// TIA Portal V16 export
// export: Created 2024-09-05T17:40:14.5392441Z, ExportSetting WithDefaults, DisplayName Totally Integrated Automation Portal, DisplayVersion V16 Update 6, DisplayName TIA Portal Version Control Interface, DisplayVersion V16 Update 2, DisplayName TIA Portal Openness, DisplayVersion V16 Update 6, DisplayName STEP 7 Professional, DisplayVersion V16 Update 6, DisplayName STEP 7 Safety, DisplayVersion V16, DisplayName WinCC Advanced, DisplayVersion V16 Update 6
TYPE "UDT_Friedrich"
// stored: IsFailsafeCompliant false
   STRUCT
      Start : Bool;
      PrgNumber : Int;
      Ready : Bool;
      Running : Bool;
      OK : Bool;
      NOK : Bool;
      H1OK : Bool;
      H2OK : Bool;
      TimeOK : Bool;
      StartError : Bool;
      LastH1 : Real;
      LastH2 : Real;
      LastTime : Real;
      LastZ1 : Real;
      Error : Bool;
      NewData : Bool;
      Z1OK : Bool;
      NewDataAfterStart : Bool;   // latched
      LastZ2 : Real;
   END_STRUCT;
END_TYPE
